Universal Robots PolyScope program: a_quarter.urp

Program a_quarter (installation=string_planes directory=/programs createdIn=5.17.3 lastSavedIn=5.17.3 robotSerialNumber=20245501435)
Calibrated DH parameters: a=[0.000154, -0.137004, -0.385524, -0.00002, 0.000092, 0]; d=[0.162441, 211.794786, -230.585024, 18.923638, 0.099786, 0.09951]; alpha=[1.569493, -0.001902, 0.003874, 1.570111, -1.570167, 0]; deltaTheta=[0, -1.242934, 1.056292, 0.186646, 0.000002, 0.000001]
InitVariablesNode
Robot Program (runOnlyOnce=false)
  MoveL speed 250 mm/s, acceleration 1200 mm/s^2 (useActiveTCP=true) feature=Plane_1
    Waypoint Waypoint_1: TCP in base x=324.752 y=765.324 z=130.385 mm, rx=-1.4944 ry=-2.2778 rz=1.1569 rad; joints [-127.056, -14.742, 33.541, -62.028, -82.973, -153.445] deg; TCP offset x=28.21 y=-96.107 z=-99.69 mm, rx=0 ry=0 rz=0 rad; feature pose in base x=325.716 y=793.387 z=118.207 mm, rx=-2.2082 ry=-0.2474 rz=-1.9195 rad
    Waypoint Waypoint_3: TCP in base x=439.971 y=533.839 z=197.07 mm, rx=-1.4944 ry=-2.2778 rz=1.1569 rad; joints [-144.985, -38.317, 71.569, -76.412, -96.031, -165.68] deg; feature pose in base x=325.716 y=793.387 z=118.207 mm, rx=-2.2082 ry=-0.2474 rz=-1.9195 rad
